SUBAPPLICATION mapping_Uebung_003a (* Subapplication Type *)
  (* Standard: 61499-2 *)
  (* Version 1.0, 2023-10-23, franz *)
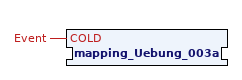
  EVENT_INPUT
    COLD;
  END_EVENT
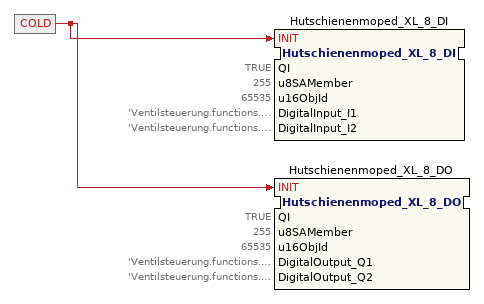
  FBS
    Hutschienenmoped_XL_8_DO : Hutschienenmoped_XL_8_DO(QI := TRUE, u8SAMember := 255, u16ObjId := 65535, DigitalOutput_Q1 := 'Ventilsteuerung.functions.F1.QX', DigitalOutput_Q2 := 'Ventilsteuerung.functions.F2.QX');
    Hutschienenmoped_XL_8_DI : Hutschienenmoped_XL_8_DI(QI := TRUE, u8SAMember := 255, u16ObjId := 65535, DigitalInput_I1 := 'Ventilsteuerung.functions.F1.IX', DigitalInput_I2 := 'Ventilsteuerung.functions.F2.IX');
  END_FBS
  EVENT_CONNECTIONS
    COLD TO Hutschienenmoped_XL_8_DI.INIT;
    COLD TO Hutschienenmoped_XL_8_DO.INIT;
  END_CONNECTIONS
END_SUBAPPLICATION
